// TIA Portal project "P4_Horak_AUT" (V16)

(* hardware
DEVICE "HMI_1"  KTP700 Basic PN
   slot 0: "HMI_1"  KTP700 Basic PN  6AV2 123-2GB03-0AX0  16.0.0.0
   slot 1: "HMI_RT_1"  KTP700 Basic PN  6AV2 123-2GB03-0AX0  16.0.0.0
   slot 5: "HMI_1.IE_CP_1"  PROFINET Interface  16.0.0.0
      slot 1: "PROFINET Interface_1"  PROFINET Interface
         slot 1: "Port_1"  Port
DEVICE "S71500/ET200MP station_1"  S7-1500 station
   slot 0: "Rail_0"  Rack  6ES7 590-1***0-0AA0
   slot 1: "PLC_1"  Unspecific CPU 1500  6ES7 5XX-XXXXX-XXXX  V2.8
*)

// ===== PLC "PLC_1"  Unspecific CPU 1500 =====

VAR_GLOBAL   // PLC tag table "Default tag table"
   "Zasobnik" AT %I0.1 : Bool;
   "Krabice" AT %I0.2 : Bool;
   "Start" AT %I0.3 : Bool;
   "Pist" AT %Q0.4 : Bool;
   "Baliky" AT %IW8 : Int;
   "DoplnitZasobnik" AT %M0.5 : Bool;
   "ZalozitKrabici" AT %M0.6 : Bool;
   "SenzorPistnice" AT %I0.4 : Bool;
END_VAR

// folder: System blocks/Program resources

DATA_BLOCK "Citac_baliku"   // DB1
{ S7_Optimized_Access := 'TRUE' }
AUTHOR : Simatic
FAMILY : IEC
NAME : CNTR
VERSION : 1.0
// stored: InstanceOfName IEC_COUNTER
"IEC_COUNTER"
BEGIN
END_DATA_BLOCK

// folder: (top level)

ORGANIZATION_BLOCK "Main"   // OB1, SCL, ProgramCycle
TITLE = "Main Program Sweep (Cycle)"
{ S7_Optimized_Access := 'TRUE' }
VERSION : 0.1
   VAR_INPUT
      Initial_Call : Bool;   // Initial call of this OB
      Remanence : Bool;   // =True, if remanent data are available
   END_VAR
BEGIN
   IF "Start" THEN //Stiskneme tlačítko start
       IF "Krabice" AND "Zasobnik" THEN //Pokud senzory detekují krabici a zasobnik
           IF "Baliky" < 6 THEN //A v krabici bude méně jak 6 balíků
               "Pist" := 1; //Píst se vysune a posune balík do krabice
           END_IF;
       END_IF;
   ELSE
       "Pist" := 0; //Výchozí poloha pístu
   END_IF;

   "Citac_baliku".CTU(CU:="Start" AND "Krabice" AND "Zasobnik", //Čítá počet balíků v krabici, dokud nebude plná
                      PV:=6, //Maximální počet balíků v krabici
                      CV=>"Baliky"); //Výstup čítače
   IF "Baliky" = 6 THEN //Pokud je krabice plná
       "ZalozitKrabici" := 1; //Zobrazí se pokyn pro výměnu krabice
   ELSE
       "ZalozitKrabici" := 0; //Pokyn se nezobrazí
   END_IF;

   IF NOT "Zasobnik" THEN //Pokud je zásobník prázdný
       "DoplnitZasobnik" := 1; //Tak se zobrazí pokyn pro doplnění
   ELSE
       "DoplnitZasobnik" := 0; //Pokyn se nezobrazí
   END_IF;
END_ORGANIZATION_BLOCK

(* ===== HMI "HMI_RT_1" =====
system functions are stored by id; their names below are inferred from use

HMI tags "Default tag table"
   "Tag_ScreenNumber" : UInt, internal

Template "Template_1" 800x480
   Button "Exit" at 714,429 size 71x50; TextOff 'Exit'; PictureOff "ExitRuntime_KTP700_Basic_PN_TR"; PictureOn "ExitRuntime_KTP700_Basic_PN_TR"
      on Release: StopRuntime(0)
   Button "Template_Button" at 614,429 size 71x50; TextOff 'Text'
   Button "Template_Button_1" at 514,429 size 71x50; TextOff 'Text'
   Button "Template_Button_2" at 414,429 size 71x50; TextOff 'Text'
   Button "Template_Button_3" at 314,429 size 71x50; TextOff 'Text'
   Button "Template_Button_4" at 214,429 size 71x50; TextOff 'Text'
   Button "Alarms" at 114,429 size 71x50; TextOff 'Alarms'; PictureOff "AlarmDisplay_KTP700_Basic_PN_TR"; PictureOn "AlarmDisplay_KTP700_Basic_PN_TR"
      on Release: function_ef3f5d25("Alarm window_Unacknowledged", -1)
   Button "Start screen" at 14,429 size 71x50; TextOff 'Start screen'; PictureOff "NavigateHome_KTP700_Basic_PN_TR"; PictureOn "NavigateHome_KTP700_Basic_PN_TR"
      on Release: ActivateScreen("Root screen", 0)
   SymbolicIOField "Symbolic_IO_Field_Screen" at 93,9 size 600x33; TextOff '0'; TextOn '1'; TextList "TextList_ScreenNames"
      ProcessValue <- "Tag_ScreenNumber"
      on Change: ActivateScreenByNumber("Tag_ScreenNumber", 0)
   DateTimeField "HmiScreenItemData" at 695,25 size 105x25
   DateTimeField "HmiScreenItemData_1" at 695,0 size 105x25
   GraphicView "Logo" at 0,0 size 91x51; Picture "Logo of HMI_1"

screen "Root screen" 800x480, template "Template_1"
   on GenerateScreen: SetTag("Tag_ScreenNumber", 1)
   TextField "Text field_1" at 350,120 size 112x28; Text 'Balící stroj'
   TextField "Text field_2" at 29,250 size 239x27; Text 'Zajistěte výchozí stav stroje'
   TextField "Text field_3" at 350,252 size 150x27; Text 'Doplňte zásobník'
   TextField "Text field_4" at 591,248 size 130x27; Text 'Založte krabici'
   Button "Button_1" at 375,347 size 105x66; TextOff 'Start'
      on Click: SetTag("Start", 1)
      on Release: SetTag("Start", 0)
   TextField "Text field_5" at 551,317 size 214x27; Text 'Počet přesunutých balíků'
   TextField "Text field_6" at 616,381 size 16x23; Text 'Text'
   IOField "I/O field_1" at 616,372 size 96x32; FormatPattern 9
*)